FUNCTION Convert_REAL_TO_BOOL : Hresult
VAR_INPUT
	in : REAL;
	out : REFERENCE TO BOOL;
END_VAR
VAR
	converted : BOOL;
END_VAR

converted := REAL_TO_BOOL(in);

IF (BOOL_TO_REAL(converted) <> in) THEN
	Convert_REAL_TO_BOOL := INCOMPATIBLE;
	RETURN;
END_IF

out := converted;

END_FUNCTION

(* stored: Version 1.1.0.1, ProductVersion 3.1.4024.12
   POU Convert_REAL_TO_BOOL: Id {dff990ba-f0e1-4615-b1b2-6139d6aebcd1}, SpecialFunc None *)
